// Mitsubishi GX Works2 project: IHW1   PLC: Q03UDE

// global labels: Global1
VAR_GLOBAL
  SS AT X50 : BOOL;
  ESTOP AT X51 : BOOL;
  CB_A AT X52 : BOOL;
  CB_B AT X53 : BOOL;
  CB_C AT X54 : BOOL;
  CB_D AT X55 : BOOL;
  LL AT Y40 : BOOL;
  XX AT Y41 : BOOL;
  TT AT Y42 : BOOL;
  PP AT Y43 : BOOL;
END_VAR

PROGRAM MAIN
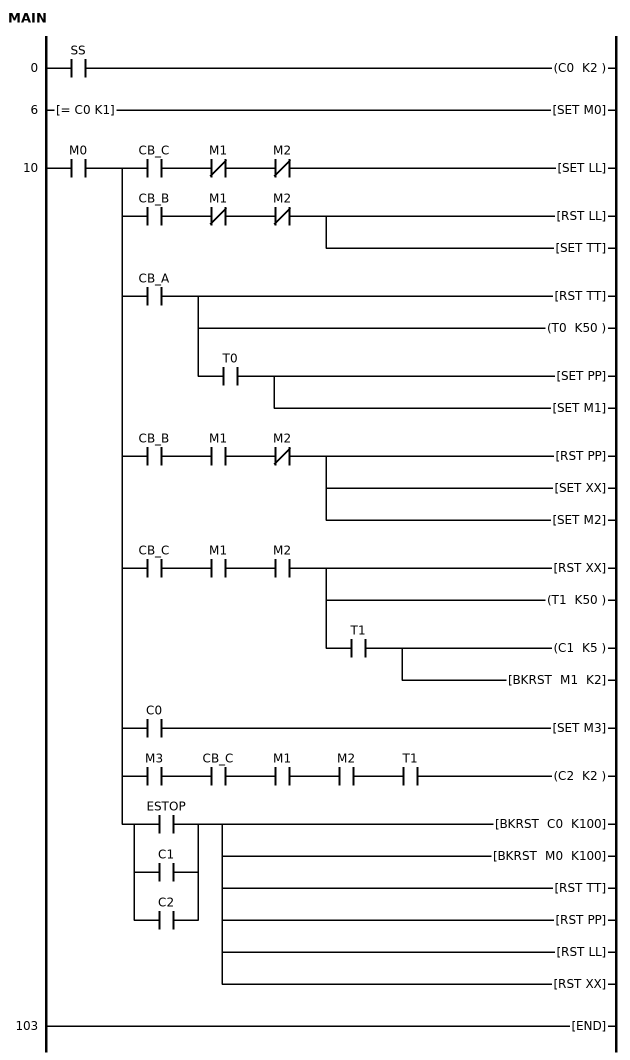
0     LD      SS
      OUT     C0 K2
6     LD=     C0 K1
      SET     M0
10    LD      M0
      MPS
      AND     CB_C
      ANI     M1
      ANI     M2
      SET     LL
      MRD
      AND     CB_B
      ANI     M1
      ANI     M2
      RST     LL
      SET     TT
      MRD
      AND     CB_A
      RST     TT
      OUT     T0 K50
      AND     T0
      SET     PP
      SET     M1
      MRD
      AND     CB_B
      AND     M1
      ANI     M2
      RST     PP
      SET     XX
      SET     M2
      MRD
      AND     CB_C
      AND     M1
      AND     M2
      RST     XX
      OUT     T1 K50
      AND     T1
      OUT     C1 K5
      BKRST   M1 K2
      MRD
      AND     C0
      SET     M3
      MRD
      AND     M3
      AND     CB_C
      AND     M1
      AND     M2
      AND     T1
      OUT     C2 K2
      MPP
      LD      ESTOP
      OR      C1
      OR      C2
      ANB
      BKRST   C0 K100
      BKRST   M0 K100
      RST     TT
      RST     PP
      RST     LL
      RST     XX
103   END
END_PROGRAM
